# EPICS autosave request: iocBoot/ioc4idHHLM/auto_settings.req
file basic_motor_settings.req P=$(P), M=m1
file basic_motor_settings.req P=$(P), M=m2
file basic_motor_settings.req P=$(P), M=m3
file basic_motor_settings.req P=$(P), M=m4
file basic_motor_settings.req P=$(P), M=m5
file basic_motor_settings.req P=$(P), M=mir:lateral
file basic_motor_settings.req P=$(P), M=mir:coarsePitch
file basic_motor_settings.req P=$(P), M=mir:curvature
